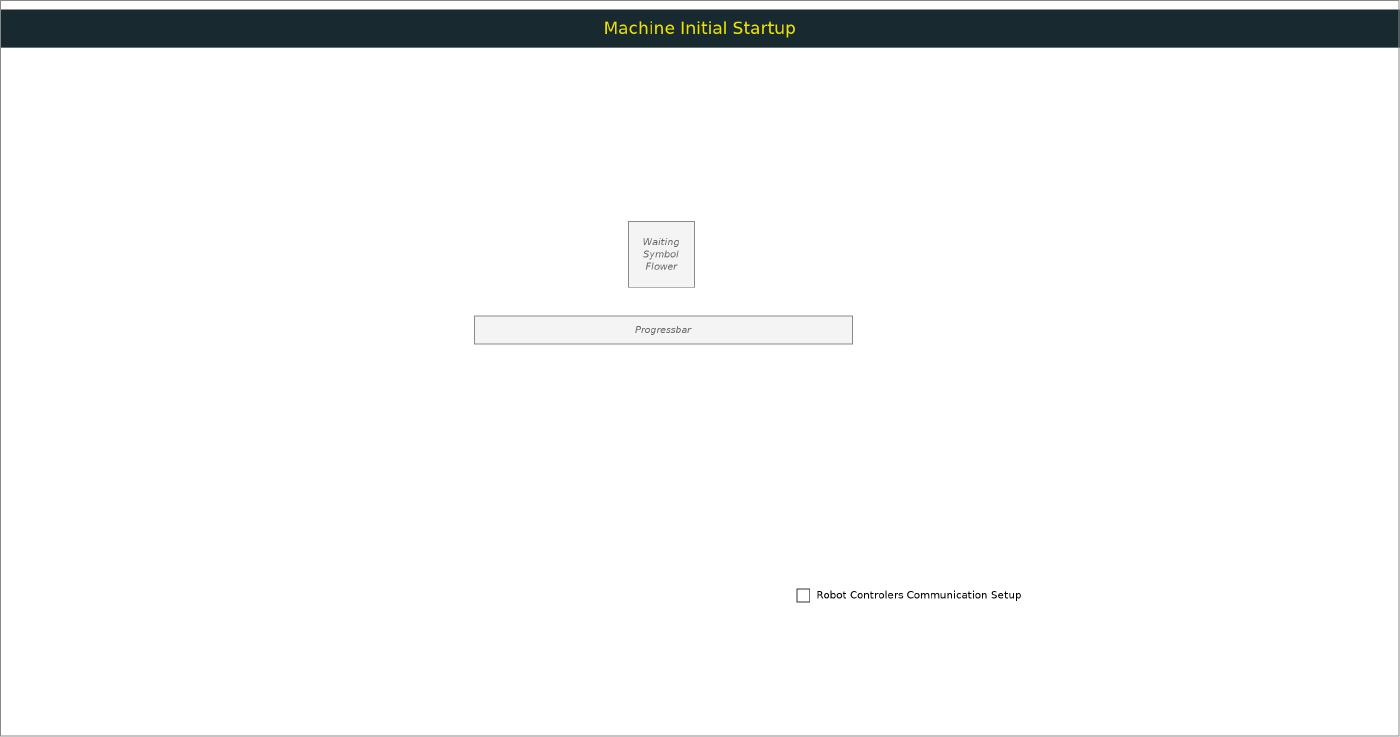
VISUALIZATION UninitializedStartUpFrame  // 1480x780
VAR_IN_OUT
	stUninitializedStartUpFrame	: ST_UninitializedStartUpFrame;
END_VAR
    Rectangle (0,10 1480x40), "Machine Initial Startup"
    Progressbar (501,334 400x30), variable: stUninitializedStartUpFrame.iProgressBar
    WaitingSymbolFlower (664,234 70x70)
    Checkbox (840,615 400x30), "Robot Controlers Communication Setup", variable: stUninitializedStartUpFrame.bCR800EtherCatInitialization
END_VISUALIZATION

(* stored: Version 1.1.0.1, ProductVersion 3.1.4024.9
   Visu UninitializedStartUpFrame: Id {7f2b516e-5a29-489c-b2e0-60a0df01cc4f} *)
